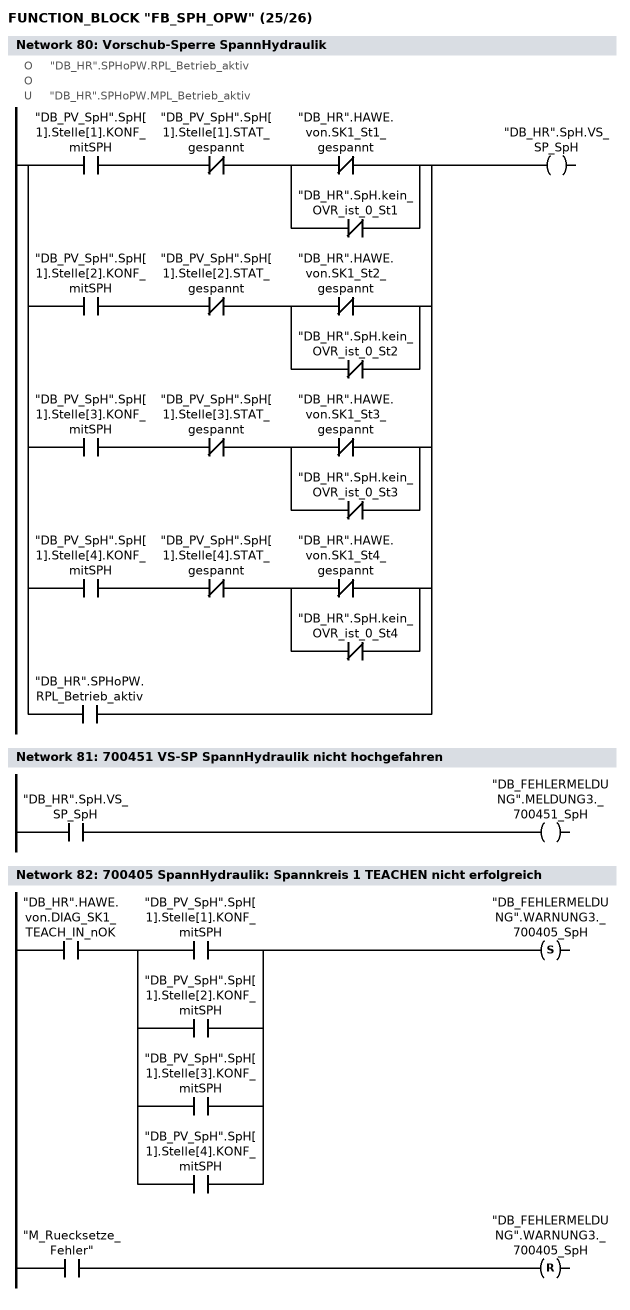
      U     "DB_PV_SpH".SpH[1].Stelle[1].KONF_mitSPH;
      UN    "DB_PV_SpH".SpH[1].Stelle[1].STAT_gespannt;
      U(    ;
      ON    "DB_HR".HAWE.von.SK1_St1_gespannt;
      ON    "DB_HR".SpH.kein_OVR_ist_0_St1;
      )     ;
      O     ;
      U     "DB_PV_SpH".SpH[1].Stelle[2].KONF_mitSPH;
      UN    "DB_PV_SpH".SpH[1].Stelle[2].STAT_gespannt;
      U(    ;
      ON    "DB_HR".HAWE.von.SK1_St2_gespannt;
      ON    "DB_HR".SpH.kein_OVR_ist_0_St2;
      )     ;
      O     ;
      U     "DB_PV_SpH".SpH[1].Stelle[3].KONF_mitSPH;
      UN    "DB_PV_SpH".SpH[1].Stelle[3].STAT_gespannt;
      U(    ;
      ON    "DB_HR".HAWE.von.SK1_St3_gespannt;
      ON    "DB_HR".SpH.kein_OVR_ist_0_St3;
      )     ;
      O     ;
      U     "DB_PV_SpH".SpH[1].Stelle[4].KONF_mitSPH;
      UN    "DB_PV_SpH".SpH[1].Stelle[4].STAT_gespannt;
      U(    ;
      ON    "DB_HR".HAWE.von.SK1_St4_gespannt;
      ON    "DB_HR".SpH.kein_OVR_ist_0_St4;
      )     ;
      O     "DB_HR".SPHoPW.RPL_Betrieb_aktiv;
      =     "DB_HR".SpH.VS_SP_SpH;
NETWORK
TITLE =700451 VS-SP SpannHydraulik nicht hochgefahren

      U     "DB_HR".SpH.VS_SP_SpH;
      =     "DB_FEHLERMELDUNG".MELDUNG3._700451_SpH;
NETWORK
TITLE =700405 SpannHydraulik: Spannkreis 1 TEACHEN nicht erfolgreich

      U     "DB_HR".HAWE.von.DIAG_SK1_TEACH_IN_nOK;
      U(    ;
      O     "DB_PV_SpH".SpH[1].Stelle[1].KONF_mitSPH;
      O     "DB_PV_SpH".SpH[1].Stelle[2].KONF_mitSPH;
      O     "DB_PV_SpH".SpH[1].Stelle[3].KONF_mitSPH;
      O     "DB_PV_SpH".SpH[1].Stelle[4].KONF_mitSPH;
      )     ;
      S     "DB_FEHLERMELDUNG".WARNUNG3._700405_SpH;
      U     "M_Ruecksetze_Fehler";
      R     "DB_FEHLERMELDUNG".WARNUNG3._700405_SpH;
      NOP   0;
NETWORK
TITLE =700414 von HAWEbox: Spannkreis 1 Druck nicht erreichbar
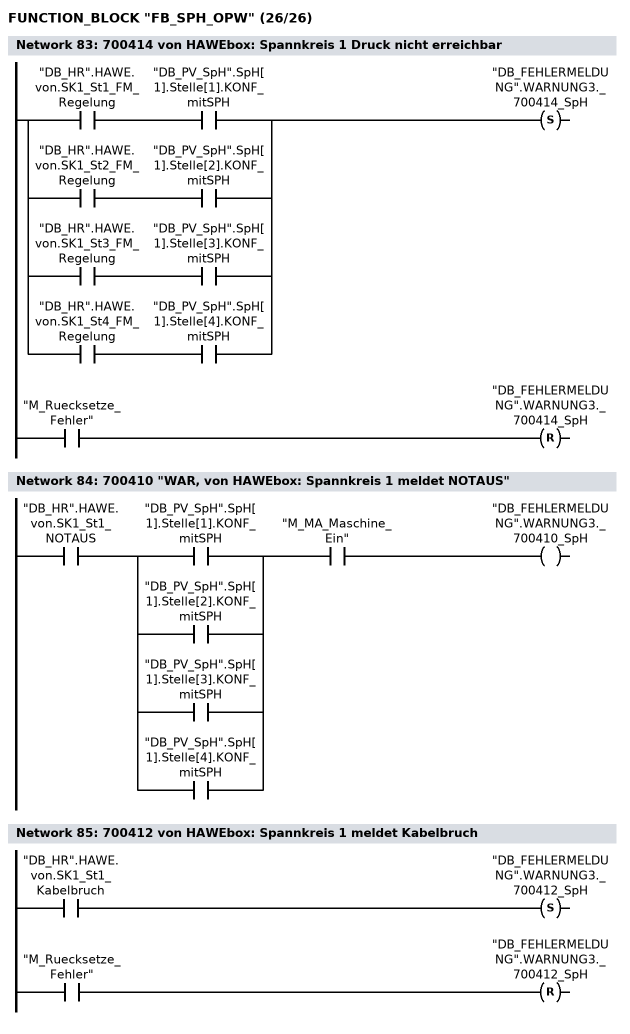

      U(    ;
      U     "DB_HR".HAWE.von.SK1_St1_FM_Regelung;
//      UN    "Tv_FM_Hawe_unterdruecken"
      U     "DB_PV_SpH".SpH[1].Stelle[1].KONF_mitSPH;
      O     ;
      U     "DB_HR".HAWE.von.SK1_St2_FM_Regelung;
//      UN    "Tv_FM_Hawe_unterdruecken"
      U     "DB_PV_SpH".SpH[1].Stelle[2].KONF_mitSPH;
      O     ;
      U     "DB_HR".HAWE.von.SK1_St3_FM_Regelung;
//      UN    "Tv_FM_Hawe_unterdruecken"
      U     "DB_PV_SpH".SpH[1].Stelle[3].KONF_mitSPH;
      O     ;
      U     "DB_HR".HAWE.von.SK1_St4_FM_Regelung;
//      UN    "Tv_FM_Hawe_unterdruecken"
      U     "DB_PV_SpH".SpH[1].Stelle[4].KONF_mitSPH;
      )     ;
      S     "DB_FEHLERMELDUNG".WARNUNG3._700414_SpH;

      U     "M_Ruecksetze_Fehler";
      R     "DB_FEHLERMELDUNG".WARNUNG3._700414_SpH;
      NOP   0;
NETWORK
TITLE =700410 "WAR, von HAWEbox: Spannkreis 1 meldet NOTAUS"

      U     "DB_HR".HAWE.von.SK1_St1_NOTAUS;
      U(    ;
      O     "DB_PV_SpH".SpH[1].Stelle[1].KONF_mitSPH;
      O     "DB_PV_SpH".SpH[1].Stelle[2].KONF_mitSPH;
      O     "DB_PV_SpH".SpH[1].Stelle[3].KONF_mitSPH;
      O     "DB_PV_SpH".SpH[1].Stelle[4].KONF_mitSPH;
      )     ;
      U     "M_MA_Maschine_Ein";
      =     "DB_FEHLERMELDUNG".WARNUNG3._700410_SpH;
NETWORK
TITLE =700412 von HAWEbox: Spannkreis 1 meldet Kabelbruch

      U     "DB_HR".HAWE.von.SK1_St1_Kabelbruch;
      S     "DB_FEHLERMELDUNG".WARNUNG3._700412_SpH;
      U     "M_Ruecksetze_Fehler";
      R     "DB_FEHLERMELDUNG".WARNUNG3._700412_SpH;
      NOP   0;
NETWORK
TITLE =Diagnose: Lebenszeichen-Überwachung

      U     "m_takt_0,5sec.";
      FP    "DB_HR".SpH.HM_PI_Takt;
      SPBN  LBZ;
      UN    "DB_HR".HAWE.an.DIAG_Lebenszeichen;
      =     "DB_HR".HAWE.an.DIAG_Lebenszeichen;
LBZ:  NOP   0;
NETWORK
TITLE =702349 "WAR, Lebenszeichen ProfiBus-HAWE-Box fehlt!"

      U(    ;
      U     "DB_HR".ABST.SpannHydraulik;
      UN    "DB_CONFIG".ABST.SPH_VORBEREITET;
      UN    "DB_HR".HAWE.von.DIAG_Lebenszeichen;
      U     "M_MA_Maschine_Ein";
      L     S5T#2S;
      SE    "Te_HAWE_Lebenszeichen";
      NOP   0;
      NOP   0;
      NOP   0;
      U     "Te_HAWE_Lebenszeichen";
      )     ;
      =     #t_LZ_HAWE_niO;
      U     #t_LZ_HAWE_niO;
      S     "DB_FEHLERMELDUNG".WARNUNG4._702349;
      UN    #t_LZ_HAWE_niO;
      U     "M_Ruecksetze_Fehler";
      R     "DB_FEHLERMELDUNG".WARNUNG4._702349;
      NOP   0;
NETWORK
TITLE =HMI-Anzeige: SpannKreis 1 Stelle 1 Istdruck
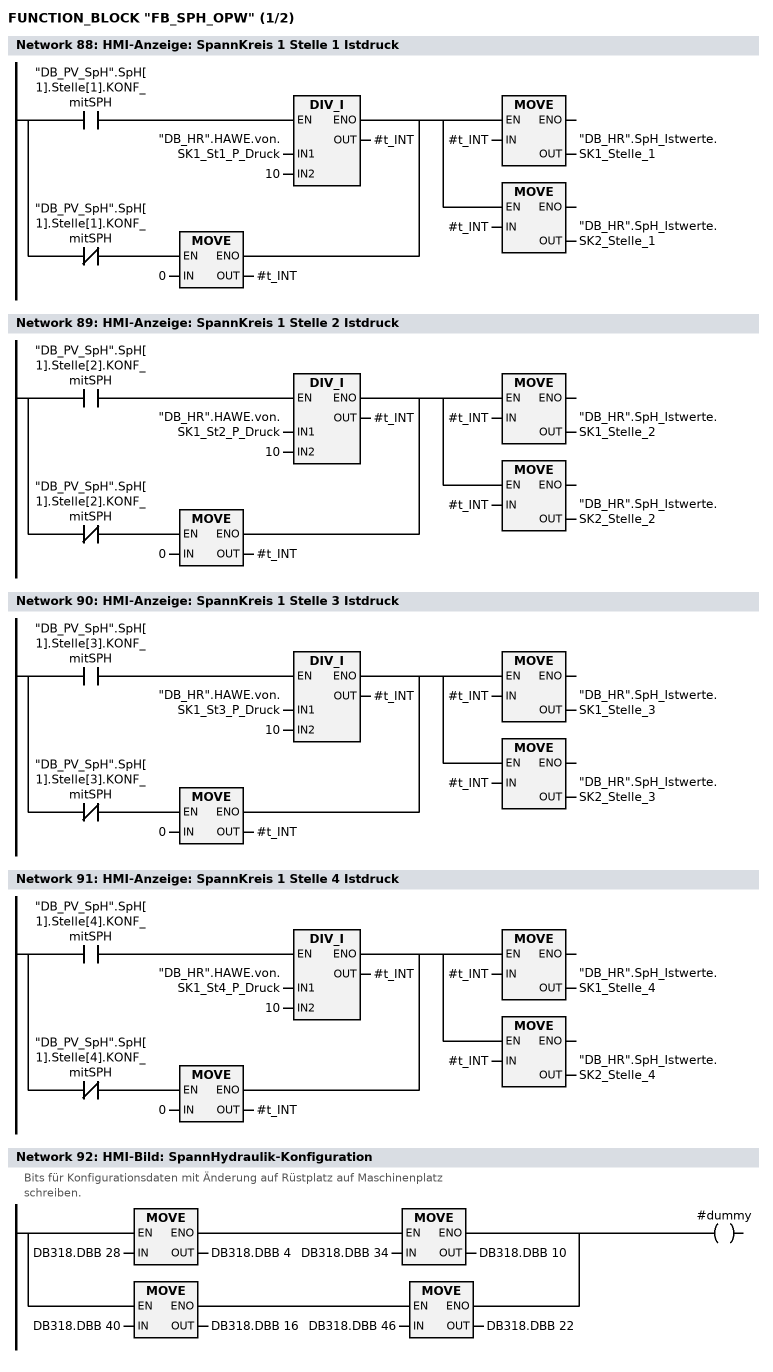

      O(    ;
      U     "DB_PV_SpH".SpH[1].Stelle[1].KONF_mitSPH;
      SPBNB _00d;
      L     "DB_HR".HAWE.von.SK1_St1_P_Druck;
      L     10;
      /I    ;
      T     #t_INT;
      UN    OV;
      SAVE  ;
      CLR   ;
_00d: U     BIE;
      )     ;
      O(    ;
      UN    "DB_PV_SpH".SpH[1].Stelle[1].KONF_mitSPH;
      SPBNB _00e;
      L     0;
      T     #t_INT;
      SET   ;
      SAVE  ;
      CLR   ;
_00e: U     BIE;
      )     ;
      =     L     16.0;
      U     L     16.0;
      SPBNB _00f;
      L     #t_INT;
      T     "DB_HR".SpH_Istwerte.SK1_Stelle_1;
_00f: NOP   0;
      U     L     16.0;
      SPBNB _010;
      L     #t_INT;
      T     "DB_HR".SpH_Istwerte.SK2_Stelle_1;
_010: NOP   0;
NETWORK
TITLE =HMI-Anzeige: SpannKreis 1 Stelle 2 Istdruck

      O(    ;
      U     "DB_PV_SpH".SpH[1].Stelle[2].KONF_mitSPH;
      SPBNB _011;
      L     "DB_HR".HAWE.von.SK1_St2_P_Druck;
      L     10;
      /I    ;
      T     #t_INT;
      UN    OV;
      SAVE  ;
      CLR   ;
_011: U     BIE;
      )     ;
      O(    ;
      UN    "DB_PV_SpH".SpH[1].Stelle[2].KONF_mitSPH;
      SPBNB _012;
      L     0;
      T     #t_INT;
      SET   ;
      SAVE  ;
      CLR   ;
_012: U     BIE;
      )     ;
      =     L     16.0;
      U     L     16.0;
      SPBNB _013;
      L     #t_INT;
      T     "DB_HR".SpH_Istwerte.SK1_Stelle_2;
_013: NOP   0;
      U     L     16.0;
      SPBNB _014;
      L     #t_INT;
      T     "DB_HR".SpH_Istwerte.SK2_Stelle_2;
_014: NOP   0;
NETWORK
TITLE =HMI-Anzeige: SpannKreis 1 Stelle 3 Istdruck

      O(    ;
      U     "DB_PV_SpH".SpH[1].Stelle[3].KONF_mitSPH;
      SPBNB _015;
      L     "DB_HR".HAWE.von.SK1_St3_P_Druck;
      L     10;
      /I    ;
      T     #t_INT;
      UN    OV;
      SAVE  ;
      CLR   ;
_015: U     BIE;
      )     ;
      O(    ;
      UN    "DB_PV_SpH".SpH[1].Stelle[3].KONF_mitSPH;
      SPBNB _016;
      L     0;
      T     #t_INT;
      SET   ;
      SAVE  ;
      CLR   ;
_016: U     BIE;
      )     ;
      =     L     16.0;
      U     L     16.0;
      SPBNB _017;
      L     #t_INT;
      T     "DB_HR".SpH_Istwerte.SK1_Stelle_3;
_017: NOP   0;
      U     L     16.0;
      SPBNB _018;
      L     #t_INT;
      T     "DB_HR".SpH_Istwerte.SK2_Stelle_3;
_018: NOP   0;
NETWORK
TITLE =HMI-Anzeige: SpannKreis 1 Stelle 4 Istdruck

      O(    ;
      U     "DB_PV_SpH".SpH[1].Stelle[4].KONF_mitSPH;
      SPBNB _019;
      L     "DB_HR".HAWE.von.SK1_St4_P_Druck;
      L     10;
      /I    ;
      T     #t_INT;
      UN    OV;
      SAVE  ;
      CLR   ;
_019: U     BIE;
      )     ;
      O(    ;
      UN    "DB_PV_SpH".SpH[1].Stelle[4].KONF_mitSPH;
      SPBNB _01a;
      L     0;
      T     #t_INT;
      SET   ;
      SAVE  ;
      CLR   ;
_01a: U     BIE;
      )     ;
      =     L     16.0;
      U     L     16.0;
      SPBNB _01b;
      L     #t_INT;
      T     "DB_HR".SpH_Istwerte.SK1_Stelle_4;
_01b: NOP   0;
      U     L     16.0;
      SPBNB _01c;
      L     #t_INT;
      T     "DB_HR".SpH_Istwerte.SK2_Stelle_4;
_01c: NOP   0;
NETWORK
TITLE =HMI-Bild: SpannHydraulik-Konfiguration
//Bits für Konfigurationsdaten mit Änderung auf Rüstplatz auf Maschinenplatz
//schreiben.
      O(    ;
      U(    ;
      L     DB318.DBB   28;
      T     DB318.DBB    4;
      SET   ;
      SAVE  ;
      CLR   ;
      U     BIE;
      )     ;
      SPBNB _01d;
      L     DB318.DBB   34;
      T     DB318.DBB   10;
      SET   ;
      SAVE  ;
      CLR   ;
_01d: U     BIE;
      )     ;
      O(    ;
      U(    ;
      L     DB318.DBB   40;
      T     DB318.DBB   16;
      SET   ;
      SAVE  ;
      CLR   ;
      U     BIE;
      )     ;
      SPBNB _01e;
      L     DB318.DBB   46;
      T     DB318.DBB   22;
      SET   ;
      SAVE  ;
      CLR   ;
_01e: U     BIE;
      )     ;
      =     #dummy;
NETWORK
TITLE =Merker SpannHydraulik-Spannen läuft
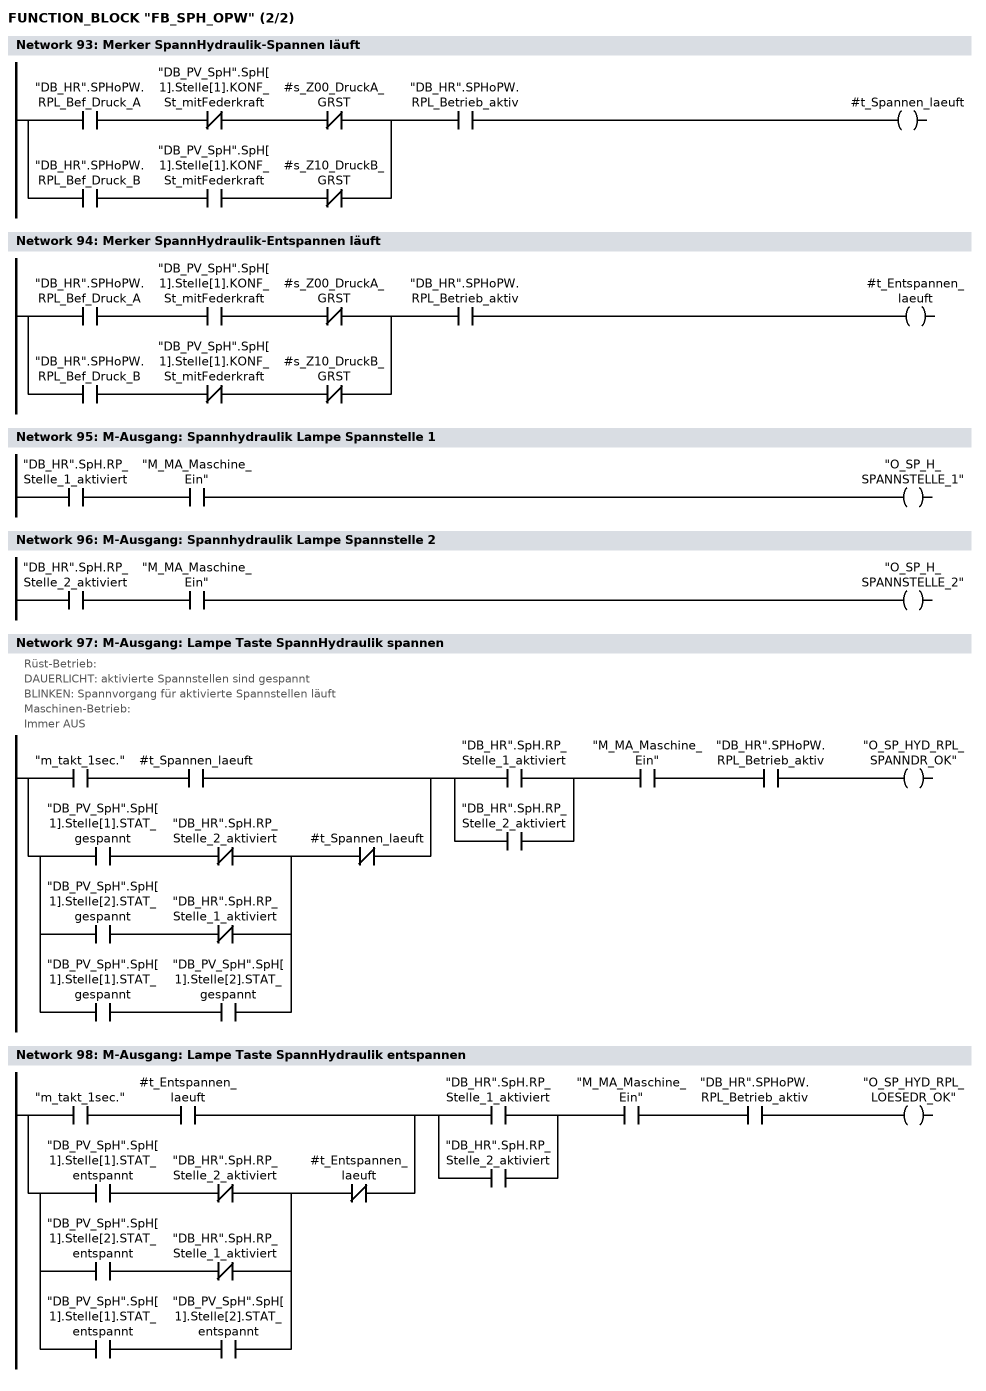

      U(    ;
      U     "DB_HR".SPHoPW.RPL_Bef_Druck_A;
      UN    "DB_PV_SpH".SpH[1].Stelle[1].KONF_St_mitFederkraft;
      UN    #s_Z00_DruckA_GRST;
      O     ;
      U     "DB_HR".SPHoPW.RPL_Bef_Druck_B;
      U     "DB_PV_SpH".SpH[1].Stelle[1].KONF_St_mitFederkraft;
      UN    #s_Z10_DruckB_GRST;
      )     ;
      U     "DB_HR".SPHoPW.RPL_Betrieb_aktiv;
      =     #t_Spannen_laeuft;
NETWORK
TITLE =Merker SpannHydraulik-Entspannen läuft

      U(    ;
      U     "DB_HR".SPHoPW.RPL_Bef_Druck_A;
      U     "DB_PV_SpH".SpH[1].Stelle[1].KONF_St_mitFederkraft;
      UN    #s_Z00_DruckA_GRST;
      O     ;
      U     "DB_HR".SPHoPW.RPL_Bef_Druck_B;
      UN    "DB_PV_SpH".SpH[1].Stelle[1].KONF_St_mitFederkraft;
      UN    #s_Z10_DruckB_GRST;
      )     ;
      U     "DB_HR".SPHoPW.RPL_Betrieb_aktiv;
      =     #t_Entspannen_laeuft;
NETWORK
TITLE =M-Ausgang: Spannhydraulik Lampe Spannstelle 1

      U     "DB_HR".SpH.RP_Stelle_1_aktiviert;
      U     "M_MA_Maschine_Ein";
      =     "O_SP_H_SPANNSTELLE_1";
NETWORK
TITLE =M-Ausgang: Spannhydraulik Lampe Spannstelle 2

      U     "DB_HR".SpH.RP_Stelle_2_aktiviert;
      U     "M_MA_Maschine_Ein";
      =     "O_SP_H_SPANNSTELLE_2";
NETWORK
TITLE =M-Ausgang: Lampe Taste SpannHydraulik spannen
//Rüst-Betrieb:
//DAUERLICHT: aktivierte Spannstellen sind gespannt
//   BLINKEN: Spannvorgang für aktivierte Spannstellen läuft
//
//Maschinen-Betrieb:
//Immer AUS
      U(    ;
      U     "m_takt_1sec.";
      U     #t_Spannen_laeuft;
      O     ;
      U(    ;
      U     "DB_PV_SpH".SpH[1].Stelle[1].STAT_gespannt;
      UN    "DB_HR".SpH.RP_Stelle_2_aktiviert;
      O     ;
      U     "DB_PV_SpH".SpH[1].Stelle[2].STAT_gespannt;
      UN    "DB_HR".SpH.RP_Stelle_1_aktiviert;
      O     ;
      U     "DB_PV_SpH".SpH[1].Stelle[1].STAT_gespannt;
      U     "DB_PV_SpH".SpH[1].Stelle[2].STAT_gespannt;
      )     ;
      UN    #t_Spannen_laeuft;
      )     ;
      U(    ;
      O     "DB_HR".SpH.RP_Stelle_1_aktiviert;
      O     "DB_HR".SpH.RP_Stelle_2_aktiviert;
      )     ;
      U     "M_MA_Maschine_Ein";
      U     "DB_HR".SPHoPW.RPL_Betrieb_aktiv;
      =     "O_SP_HYD_RPL_SPANNDR_OK";
NETWORK
TITLE =M-Ausgang: Lampe Taste SpannHydraulik entspannen

      U(    ;
      U     "m_takt_1sec.";
      U     #t_Entspannen_laeuft;
      O     ;
      U(    ;
      U     "DB_PV_SpH".SpH[1].Stelle[1].STAT_entspannt;
      UN    "DB_HR".SpH.RP_Stelle_2_aktiviert;

      O     ;
      U     "DB_PV_SpH".SpH[1].Stelle[2].STAT_entspannt;
      UN    "DB_HR".SpH.RP_Stelle_1_aktiviert;
      O     ;
      U     "DB_PV_SpH".SpH[1].Stelle[1].STAT_entspannt;
      U     "DB_PV_SpH".SpH[1].Stelle[2].STAT_entspannt;
      )     ;
      UN    #t_Entspannen_laeuft;
      )     ;
      U(    ;
      O     "DB_HR".SpH.RP_Stelle_1_aktiviert;
      O     "DB_HR".SpH.RP_Stelle_2_aktiviert;
      )     ;
      U     "M_MA_Maschine_Ein";
      U     "DB_HR".SPHoPW.RPL_Betrieb_aktiv;
      =     "O_SP_HYD_RPL_LOESEDR_OK";
END_FUNCTION_BLOCK

